Fanuc KAREL source: kf00084.KL

-- PROVISIONAL review KL for V1013-1; original PC SHA256 de2735af5328cbe9e21ba3e75d42809c49298b883c39388c80d69c7ebe71ed6a
-- Incomplete behavior may be omitted. Consult companion uncertainty JSON. Do not deploy.
PROGRAM KF00084
%NOLOCKGROUP
VAR
  I : INTEGER
  J : INTEGER
  X : REAL
  Y : REAL
  B : BOOLEAN
  C : BOOLEAN
  TXT : STRING[80]
  TXT2 : STRING[80]
  STATUS : INTEGER
-- UNRESOLVED_DECL AI type=002010
-- UNRESOLVED_DECL BI type=002010
-- UNRESOLVED_DECL P type=000102
-- UNRESOLVED_DECL JP type=000199
-- UNRESOLVED_DECL PF type=000101
-- UNRESOLVED_DECL V1 type=000013
-- UNRESOLVED_DECL V2 type=000013
BEGIN
  -- UNRESOLVED_PC offsets 5-26; opcodes 27,27,9C,27,9C,27,9D,76,7E,4A
  -- UNRESOLVED_PC offsets 31-35; opcodes 7F
END KF00084
